# EPICS substitutions: ioc/PSCApp/Db/inp_waveform.substitutions
file db/inp_waveform.db {
    pattern {INP_CHANNEL_NUMBER}
        {"1"}
}
